// TIA Portal V16 export
// export: Created 2024-09-05T17:39:18.2304179Z, ExportSetting WithDefaults, DisplayName Totally Integrated Automation Portal, DisplayVersion V16 Update 6, DisplayName TIA Portal Version Control Interface, DisplayVersion V16 Update 2, DisplayName TIA Portal Openness, DisplayVersion V16 Update 6, DisplayName STEP 7 Professional, DisplayVersion V16 Update 6, DisplayName STEP 7 Safety, DisplayVersion V16, DisplayName WinCC Advanced, DisplayVersion V16 Update 6
DATA_BLOCK "CycleTimeMeas_Fitting1_DB"   // DB31
VERSION : 0.1
// stored: AutoNumber true, DBAccessibleFromOPCUA true, InstanceOfName CycleTimeMeas, InstanceOfType FB
"CycleTimeMeas"
   // VAR_INPUT
   //    StartCycle : Bool := FALSE;
   //    ResetHistory : Bool := FALSE;
   // END_VAR
   // VAR
   //    ActualTime : Time := T#0MS;
   //    LastTime : Time := T#12S_830MS;
   //    edge2 : Bool := FALSE;
   //    edge1 : Bool := FALSE;
   //    Suma : DInt := 35860;
   //    Count : DInt := 3;
   //    Max : Time := T#13S_176MS;
   //    Min : Time := T#9S_854MS;
   //    Average : Time := T#11S_953MS;
   //    IEC_Timer_0_Instance { S7_SetPoint := 'True'} : TON_TIME;
   //    History : Array[1..20] of Time;
   //    NewTime : Bool := FALSE;
   // END_VAR
BEGIN
   IEC_Timer_0_Instance.PT := T#8M_20S;
   IEC_Timer_0_Instance.IN := FALSE;
   History[1] := T#12S_830MS;
   History[2] := T#13S_176MS;
   History[3] := T#9S_854MS;
   History[4..20] := T#0MS;
END_DATA_BLOCK
